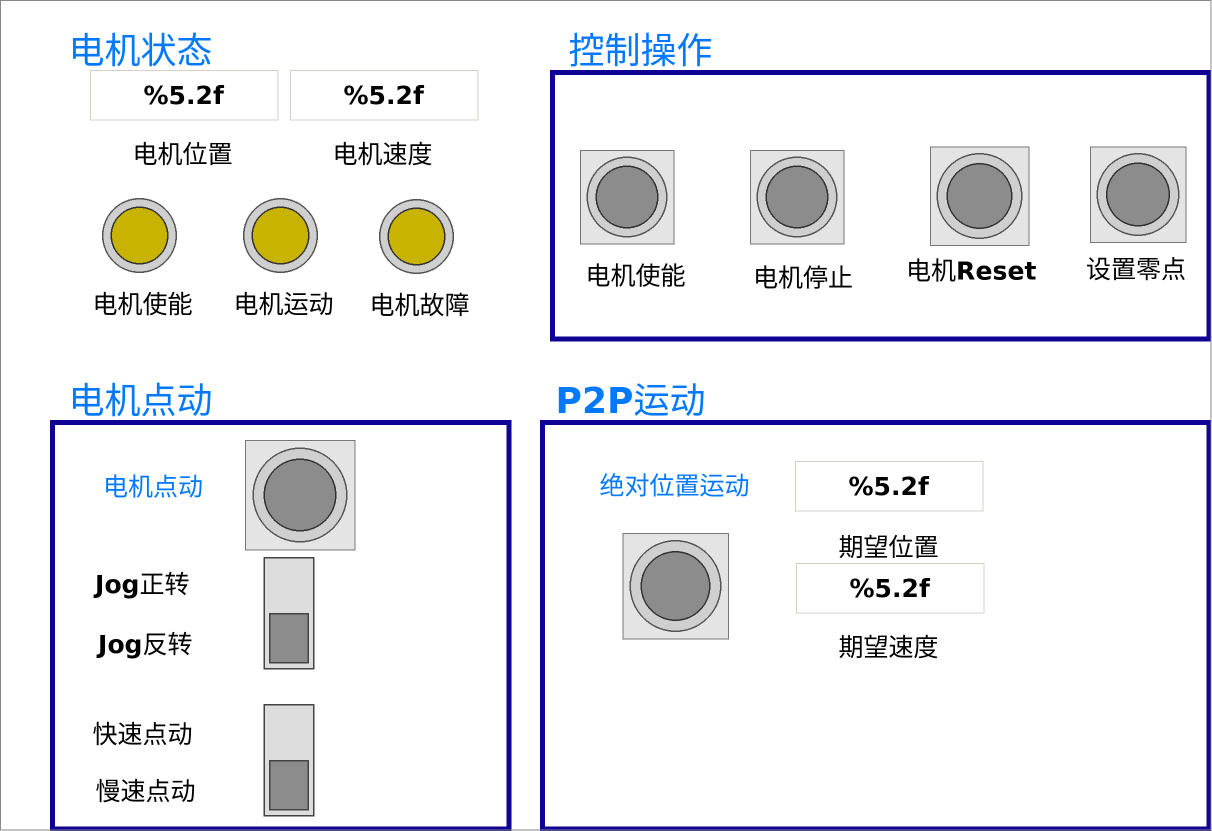
VISUALIZATION Visualization  // 1212x831
    Lamp1 (96,190 87x91), variable: Main.motor_state.is_power_ready, style: Lamp-Lamp1-Yellow
    Label (50,270 185x68), "电机使能"
    Textfield (90,70 188x50), "%5.2f", text variable: Main.motor_data.motor_position
    Label (90,120 185x68), "电机位置"
    Textfield (290,70 188x50), "%5.2f", text variable: Main.motor_data.motor_velocity
    Label (290,120 185x68), "电机速度"
    Lamp1 (237,190 87x91), variable: Main.motor_state.is_motor_moving, style: Lamp-Lamp1-Yellow
    Label (191,270 185x68), "电机运动"
    Label (327,271 185x68), "电机故障"
    Lamp1 (373,191 87x91), variable: Main.motor_state.is_motor_error, style: Lamp-Lamp1-Yellow
    Label (40,20 201x61), "电机状态"
    Rectangle (550,70 661x271)
    Label (560,250 151x51), "电机使能"
    PushSwitchLed (750,140 94x114), variable: Main.motor_param.is_motor_stop, behaviour: TAP, style: Switch-PushSwitchLed-Gray
    Label (730,250 146x55), "电机停止"
    PushSwitchLed (930,140 99x112), variable: Main.motor_param.is_motor_reset, behaviour: TAP, style: Switch-PushSwitchLed-Gray
    Label (890,250 163x41), "电机Reset"
    PushSwitchLed (1090,140 96x109), variable: Main.motor_param.is_set_pos_zero, behaviour: TAP, style: Switch-PushSwitchLed-Gray
    Label (1060,250 152x38), "设置零点"
    PushSwitchLed (580,140 94x114), variable: Main.motor_param.is_motor_power_on, behaviour: TOGGLE, style: Switch-PushSwitchLed-Gray
    Label (540,20 201x61), "控制操作"
    Rectangle (50,420 461x411)
    Label (53,610 185x68), "Jog反转"
    DipSwitch (232,557 114x112), variable: Main.motor_param.jog_direction, behaviour: TOGGLE, style: Switch-DipSwitch-Gray
    Label (50,550 185x68), "Jog正转"
    PushSwitchLed (240,440 120x110), variable: Main.motor_param.is_jog_start, behaviour: TAP, style: Switch-PushSwitchLed-Gray
    Label (90,420 126x133), "电机点动"
    Label (50,700 185x68), "快速点动"
    Label (53,757 185x68), "慢速点动"
    DipSwitch (232,704 114x112), variable: Main.motor_param.jog_mode, behaviour: TOGGLE, style: Switch-DipSwitch-Gray
    Label (40,370 201x61), "电机点动"
    Rectangle (540,420 671x411)
    Textfield (795,461 188x50), "%5.2f", text variable: Main.motor_param.move_abs_target_position
        OnMouseClick: write the text variable via Default
    Label (796,513 185x68), "期望位置"
    Label (796,613 185x68), "期望速度"
    Textfield (796,563 188x50), "%5.2f", text variable: Main.motor_param.move_vel
        OnMouseClick: write the text variable via Default
    PushSwitchLed (616,533 119x106), variable: Main.motor_param.is_motor_moving_abs, behaviour: TAP, style: Switch-PushSwitchLed-Gray
    Label (550,430 249x111), "绝对位置运动"
    Label (530,370 201x61), "P2P运动"
END_VISUALIZATION

(* stored: Version 1.1.0.1, ProductVersion 3.1.4024.11
   Visu Visualization: Id {4f144a4b-bbfd-40b9-896b-b5558eeb16b4} *)
